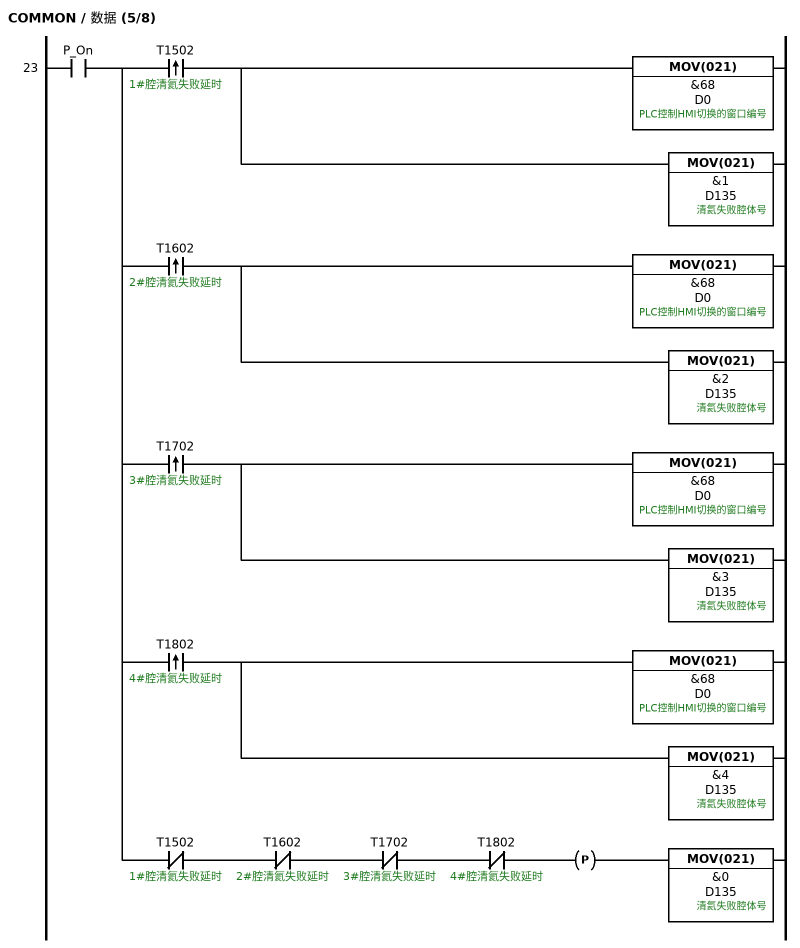
; [picture p432: COMMON / 数据, rungs 23-23]
; rung 23
LD P_On
OUT TR0
@AND T1502  ; 1#腔清氦失败延时
MOV(021) &68 D0  ; PLC控制HMI切换的窗口编号
MOV(021) &1 D135  ; 清氦失败腔体号
LD TR0
@AND T1602  ; 2#腔清氦失败延时
MOV(021) &68 D0  ; PLC控制HMI切换的窗口编号
MOV(021) &2 D135  ; 清氦失败腔体号
LD TR0
@AND T1702  ; 3#腔清氦失败延时
MOV(021) &68 D0  ; PLC控制HMI切换的窗口编号
MOV(021) &3 D135  ; 清氦失败腔体号
LD TR0
@AND T1802  ; 4#腔清氦失败延时
MOV(021) &68 D0  ; PLC控制HMI切换的窗口编号
MOV(021) &4 D135  ; 清氦失败腔体号
LD TR0
ANDNOT T1502  ; 1#腔清氦失败延时
ANDNOT T1602  ; 2#腔清氦失败延时
ANDNOT T1702  ; 3#腔清氦失败延时
ANDNOT T1802  ; 4#腔清氦失败延时
UP(521)
MOV(021) &0 D135  ; 清氦失败腔体号

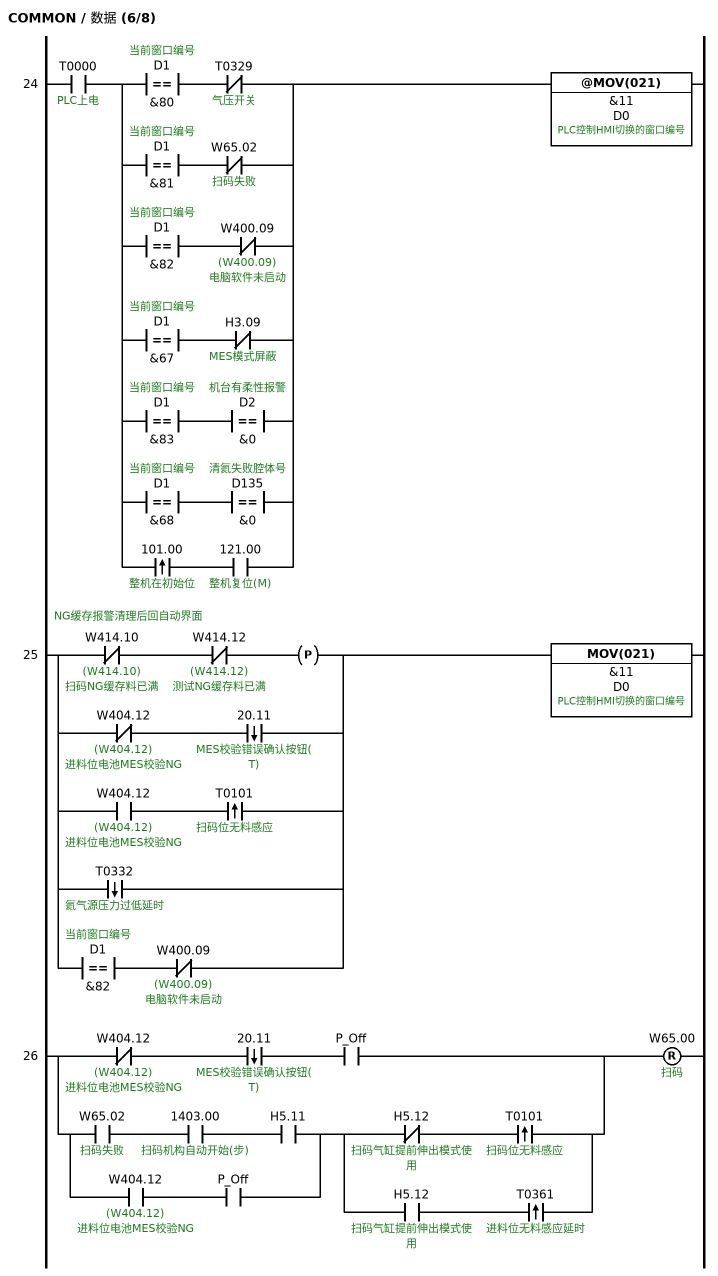
; rung 24
LD T0000  ; PLC上电
LD=(300) D1 &80  ; 当前窗口编号
ANDNOT T0329  ; 气压开关
LD=(300) D1 &81  ; 当前窗口编号
ANDNOT W65.02  ; 扫码失败
ORLD
LD=(300) D1 &82  ; 当前窗口编号
ANDNOT W400.09  ; (W400.09) 电脑软件未启动
ORLD
LD=(300) D1 &67  ; 当前窗口编号
ANDNOT H3.09  ; MES模式屏蔽
ORLD
LD=(300) D1 &83  ; 当前窗口编号
AND=(300) D2 &0  ; 机台有柔性报警
ORLD
LD=(300) D1 &68  ; 当前窗口编号
AND=(300) D135 &0  ; 清氦失败腔体号
ORLD
@LD 101.00  ; 整机在初始位
AND 121.00  ; 整机复位(M)
ORLD
ANDLD
@MOV(021) &11 D0  ; PLC控制HMI切换的窗口编号
; rung 25: NG缓存报警清理后回自动界面
LDNOT W414.10  ; (W414.10) 扫码NG缓存料已满
ANDNOT W414.12  ; (W414.12) 测试NG缓存料已满
UP(521)
LDNOT W404.12  ; (W404.12) 进料位电池MES校验NG
%AND 20.11  ; MES校验错误确认按钮(T)
ORLD
LD W404.12  ; (W404.12) 进料位电池MES校验NG
@AND T0101  ; 扫码位无料感应
ORLD
%OR T0332  ; 氦气源压力过低延时
LD=(300) D1 &82  ; 当前窗口编号
ANDNOT W400.09  ; (W400.09) 电脑软件未启动
ORLD
MOV(021) &11 D0  ; PLC控制HMI切换的窗口编号
; rung 26
LDNOT W404.12  ; (W404.12) 进料位电池MES校验NG
%AND 20.11  ; MES校验错误确认按钮(T)
AND P_Off
LD W65.02  ; 扫码失败
AND 1403.00  ; 扫码机构自动开始(步)
AND H5.11
LD W404.12  ; (W404.12) 进料位电池MES校验NG
AND P_Off
ORLD
LDNOT H5.12  ; 扫码气缸提前伸出模式使用
@AND T0101  ; 扫码位无料感应
LD H5.12  ; 扫码气缸提前伸出模式使用
@AND T0361  ; 进料位无料感应延时
ORLD
ANDLD
ORLD
RSET W65.00  ; 扫码

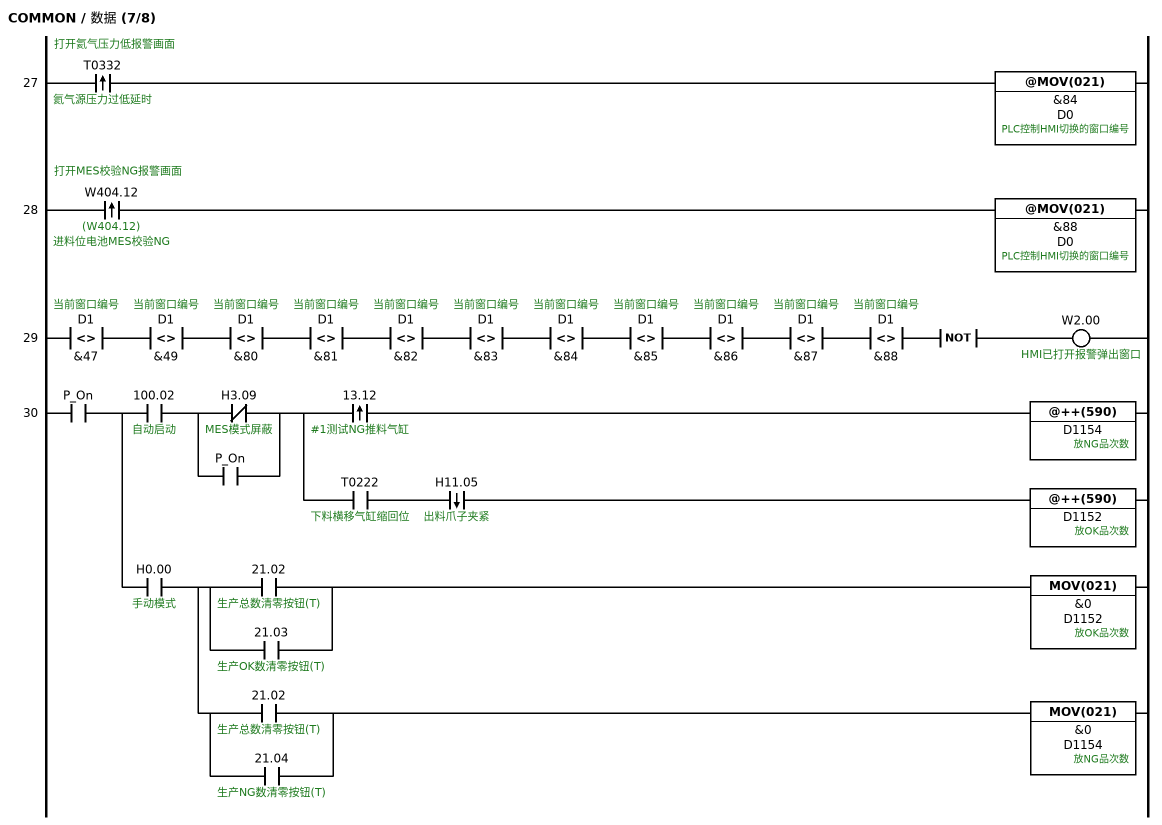
; rung 27: 打开氦气压力低报警画面
@LD T0332  ; 氦气源压力过低延时
@MOV(021) &84 D0  ; PLC控制HMI切换的窗口编号
; rung 28: 打开MES校验NG报警画面
@LD W404.12  ; (W404.12) 进料位电池MES校验NG
@MOV(021) &88 D0  ; PLC控制HMI切换的窗口编号
; rung 29
LD<>(305) D1 &47  ; 当前窗口编号
AND<>(305) D1 &49  ; 当前窗口编号
AND<>(305) D1 &80  ; 当前窗口编号
AND<>(305) D1 &81  ; 当前窗口编号
AND<>(305) D1 &82  ; 当前窗口编号
AND<>(305) D1 &83  ; 当前窗口编号
AND<>(305) D1 &84  ; 当前窗口编号
AND<>(305) D1 &85  ; 当前窗口编号
AND<>(305) D1 &86  ; 当前窗口编号
AND<>(305) D1 &87  ; 当前窗口编号
AND<>(305) D1 &88  ; 当前窗口编号
NOT(520)
OUT W2.00  ; HMI已打开报警弹出窗口
; rung 30
LD P_On
OUT TR0
AND 100.02  ; 自动启动
LDNOT H3.09  ; MES模式屏蔽
OR P_On
ANDLD
OUT TR1
@AND 13.12  ; #1测试NG推料气缸
@++(590) D1154  ; 放NG品次数
LD TR1
AND T0222  ; 下料横移气缸缩回位
%AND H11.05  ; 出料爪子夹紧
@++(590) D1152  ; 放OK品次数
LD TR0
AND H0.00  ; 手动模式
OUT TR0
LD 21.02  ; 生产总数清零按钮(T)
OR 21.03  ; 生产OK数清零按钮(T)
ANDLD
MOV(021) &0 D1152  ; 放OK品次数
LD TR0
LD 21.02  ; 生产总数清零按钮(T)
OR 21.04  ; 生产NG数清零按钮(T)
ANDLD
MOV(021) &0 D1154  ; 放NG品次数

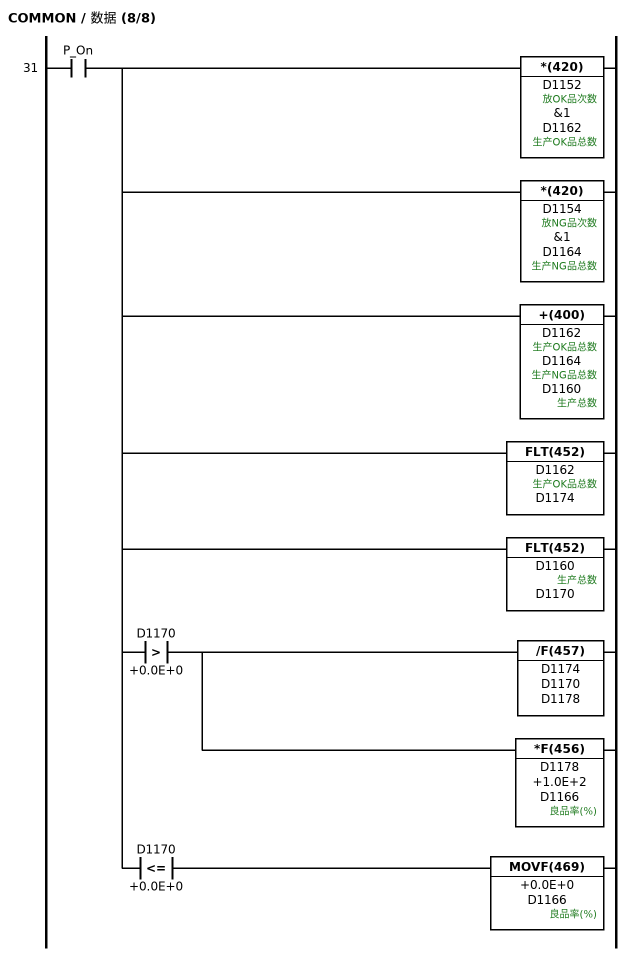
; rung 31
LD P_On
OUT TR0
*(420) D1152 &1 D1162  ; 放OK品次数, 生产OK品总数
*(420) D1154 &1 D1164  ; 放NG品次数, 生产NG品总数
+(400) D1162 D1164 D1160  ; 生产OK品总数, 生产NG品总数, 生产总数
FLT(452) D1162 D1174  ; 生产OK品总数
FLT(452) D1160 D1170  ; 生产总数
AND>F(333) D1170 +0.0E+0
/F(457) D1174 D1170 D1178
*F(456) D1178 +1.0E+2 D1166  ; 良品率(%)
LD TR0
AND<=F(332) D1170 +0.0E+0
MOVF(469) +0.0E+0 D1166  ; 良品率(%)

### Section 报警

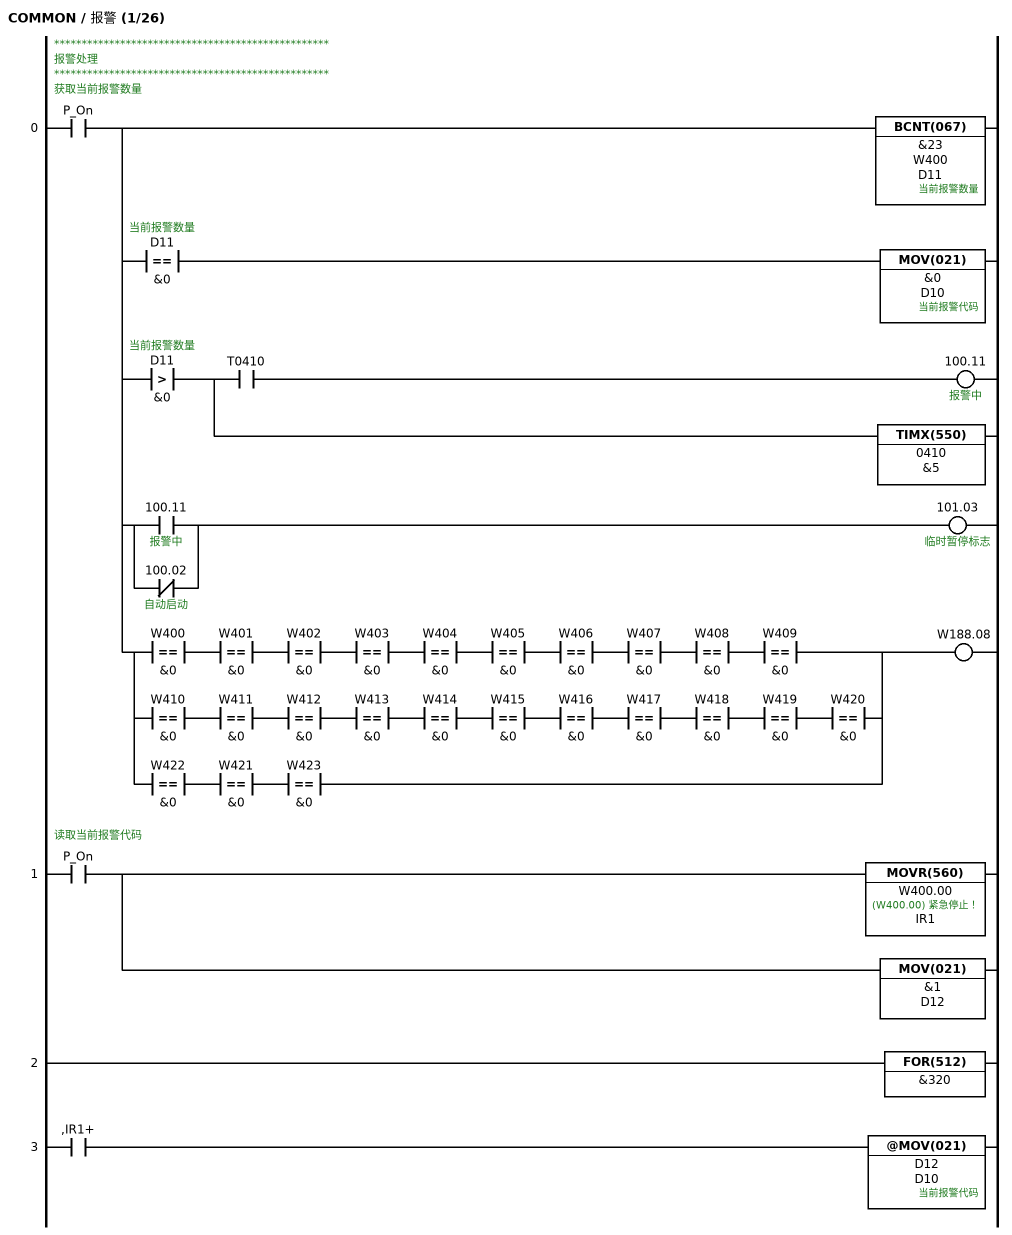
; rung 0: ************************************************** / 报警处理 / ************************************************** / 获取当前报警数量
LD P_On
OUT TR0
BCNT(067) &23 W400 D11  ; 当前报警数量
AND=(300) D11 &0  ; 当前报警数量
MOV(021) &0 D10  ; 当前报警代码
LD TR0
AND>(320) D11 &0  ; 当前报警数量
OUT TR1
AND T0410
OUT 100.11  ; 报警中
LD TR1
TIMX(550) 0410 &5
LD TR0
LD 100.11  ; 报警中
ORNOT 100.02  ; 自动启动
ANDLD
OUT 101.03  ; 临时暂停标志
LD TR0
LD=(300) W400 &0
AND=(300) W401 &0
AND=(300) W402 &0
AND=(300) W403 &0
AND=(300) W404 &0
AND=(300) W405 &0
AND=(300) W406 &0
AND=(300) W407 &0
AND=(300) W408 &0
AND=(300) W409 &0
LD=(300) W410 &0
AND=(300) W411 &0
AND=(300) W412 &0
AND=(300) W413 &0
AND=(300) W414 &0
AND=(300) W415 &0
AND=(300) W416 &0
AND=(300) W417 &0
AND=(300) W418 &0
AND=(300) W419 &0
AND=(300) W420 &0
ORLD
LD=(300) W422 &0
AND=(300) W421 &0
AND=(300) W423 &0
ORLD
ANDLD
OUT W188.08
; rung 1: 读取当前报警代码
LD P_On
MOVR(560) W400.00 IR1  ; (W400.00) 紧急停止！
MOV(021) &1 D12
; rung 2
FOR(512) &320
; rung 3
LD ,IR1+
@MOV(021) D12 D10  ; 当前报警代码

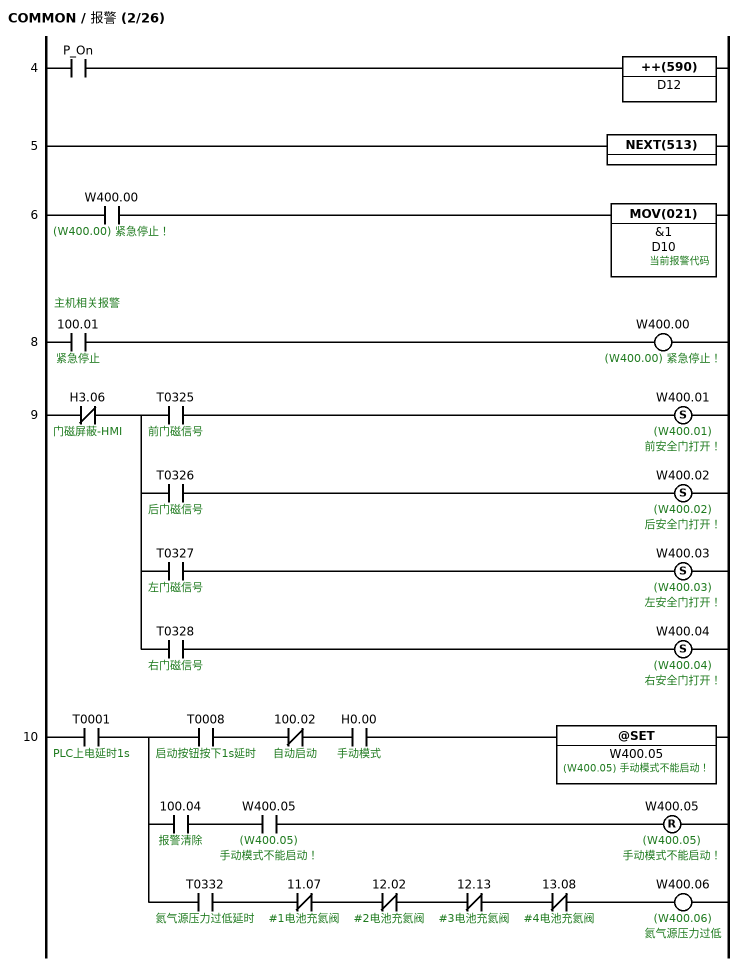
; rung 4
LD P_On
++(590) D12
; rung 5
NEXT(513)
; rung 6
LD W400.00  ; (W400.00) 紧急停止！
MOV(021) &1 D10  ; 当前报警代码
; rung 7: ************************************************************************** / 报警处理 / **************************************************************************
; rung 8: 主机相关报警
LD 100.01  ; 紧急停止
OUT W400.00  ; (W400.00) 紧急停止！
; rung 9
LDNOT H3.06  ; 门磁屏蔽-HMI
OUT TR0
AND T0325  ; 前门磁信号
SET W400.01  ; (W400.01) 前安全门打开！
LD TR0
AND T0326  ; 后门磁信号
SET W400.02  ; (W400.02) 后安全门打开！
LD TR0
AND T0327  ; 左门磁信号
SET W400.03  ; (W400.03) 左安全门打开！
LD TR0
AND T0328  ; 右门磁信号
SET W400.04  ; (W400.04) 右安全门打开！
; rung 10
LD T0001  ; PLC上电延时1s
OUT TR0
AND T0008  ; 启动按钮按下1s延时
ANDNOT 100.02  ; 自动启动
AND H0.00  ; 手动模式
@SET W400.05  ; (W400.05) 手动模式不能启动！
LD TR0
AND 100.04  ; 报警清除
AND W400.05  ; (W400.05) 手动模式不能启动！
RSET W400.05  ; (W400.05) 手动模式不能启动！
LD TR0
AND T0332  ; 氦气源压力过低延时
ANDNOT 11.07  ; #1电池充氦阀
ANDNOT 12.02  ; #2电池充氦阀
ANDNOT 12.13  ; #3电池充氦阀
ANDNOT 13.08  ; #4电池充氦阀
OUT W400.06  ; (W400.06) 氦气源压力过低

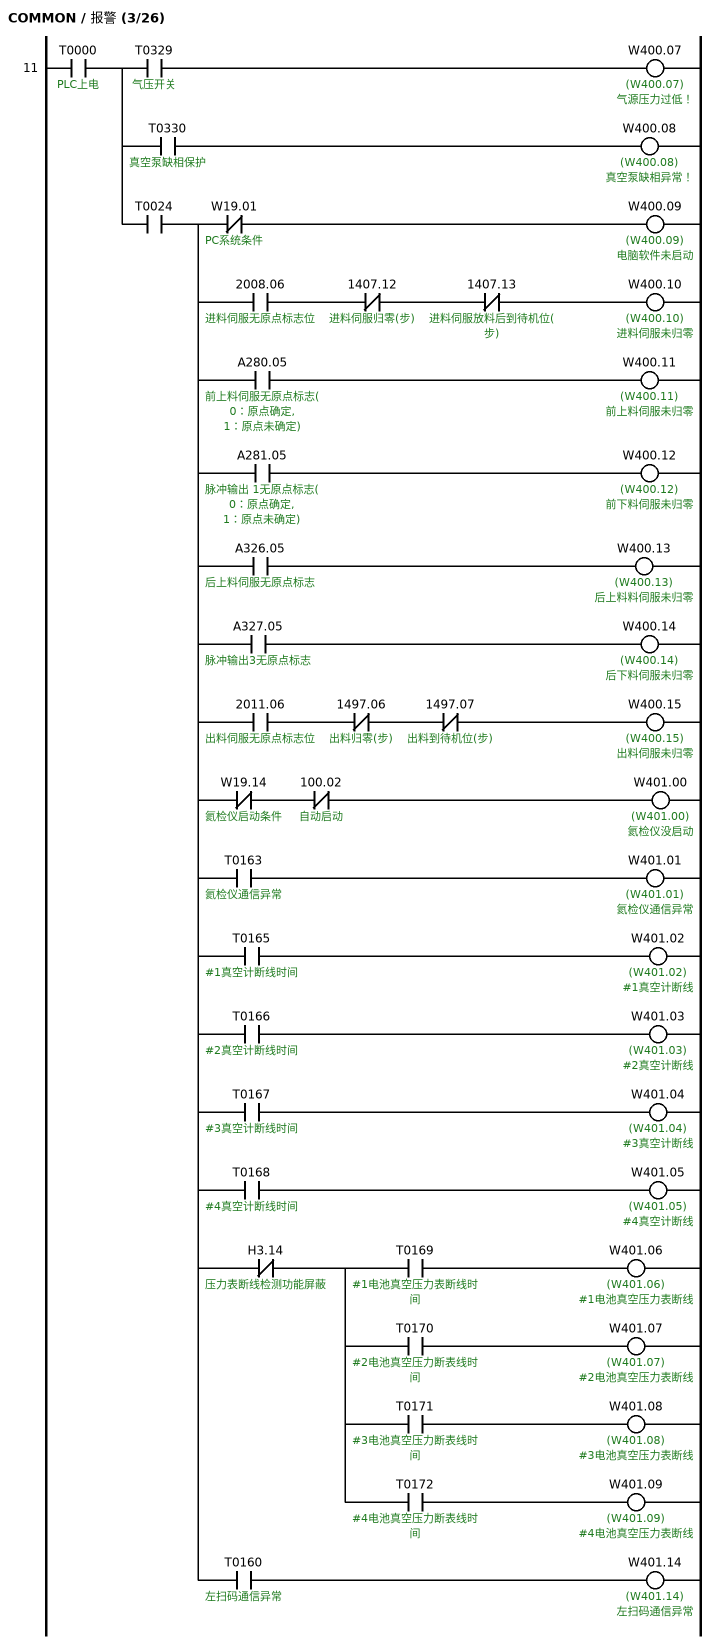
; rung 11
LD T0000  ; PLC上电
OUT TR0
AND T0329  ; 气压开关
OUT W400.07  ; (W400.07) 气源压力过低！
LD TR0
AND T0330  ; 真空泵缺相保护
OUT W400.08  ; (W400.08) 真空泵缺相异常！
LD TR0
AND T0024
OUT TR0
ANDNOT W19.01  ; PC系统条件
OUT W400.09  ; (W400.09) 电脑软件未启动
LD TR0
AND 2008.06  ; 进料伺服无原点标志位
ANDNOT 1407.12  ; 进料伺服归零(步)
ANDNOT 1407.13  ; 进料伺服放料后到待机位(步)
OUT W400.10  ; (W400.10) 进料伺服未归零
LD TR0
AND A280.05  ; 前上料伺服无原点标志(0：原点确定,1：原点未确定)
OUT W400.11  ; (W400.11) 前上料伺服未归零
LD TR0
AND A281.05  ; 脉冲输出 1无原点标志(0：原点确定,1：原点未确定)
OUT W400.12  ; (W400.12) 前下料伺服未归零
LD TR0
AND A326.05  ; 后上料伺服无原点标志
OUT W400.13  ; (W400.13) 后上料料伺服未归零
LD TR0
AND A327.05  ; 脉冲输出3无原点标志
OUT W400.14  ; (W400.14) 后下料伺服未归零
LD TR0
AND 2011.06  ; 出料伺服无原点标志位
ANDNOT 1497.06  ; 出料归零(步)
ANDNOT 1497.07  ; 出料到待机位(步)
OUT W400.15  ; (W400.15) 出料伺服未归零
LD TR0
ANDNOT W19.14  ; 氦检仪启动条件
ANDNOT 100.02  ; 自动启动
OUT W401.00  ; (W401.00) 氦检仪没启动
LD TR0
AND T0163  ; 氦检仪通信异常
OUT W401.01  ; (W401.01) 氦检仪通信异常
LD TR0
AND T0165  ; #1真空计断线时间
OUT W401.02  ; (W401.02) #1真空计断线
LD TR0
AND T0166  ; #2真空计断线时间
OUT W401.03  ; (W401.03) #2真空计断线
LD TR0
AND T0167  ; #3真空计断线时间
OUT W401.04  ; (W401.04) #3真空计断线
LD TR0
AND T0168  ; #4真空计断线时间
OUT W401.05  ; (W401.05) #4真空计断线
LD TR0
ANDNOT H3.14  ; 压力表断线检测功能屏蔽
OUT TR1
AND T0169  ; #1电池真空压力表断线时间
OUT W401.06  ; (W401.06) #1电池真空压力表断线
LD TR1
AND T0170  ; #2电池真空压力断表线时间
OUT W401.07  ; (W401.07) #2电池真空压力表断线
LD TR1
AND T0171  ; #3电池真空压力断表线时间
OUT W401.08  ; (W401.08) #3电池真空压力表断线
LD TR1
AND T0172  ; #4电池真空压力断表线时间
OUT W401.09  ; (W401.09) #4电池真空压力表断线
LD TR0
AND T0160  ; 左扫码通信异常
OUT W401.14  ; (W401.14) 左扫码通信异常

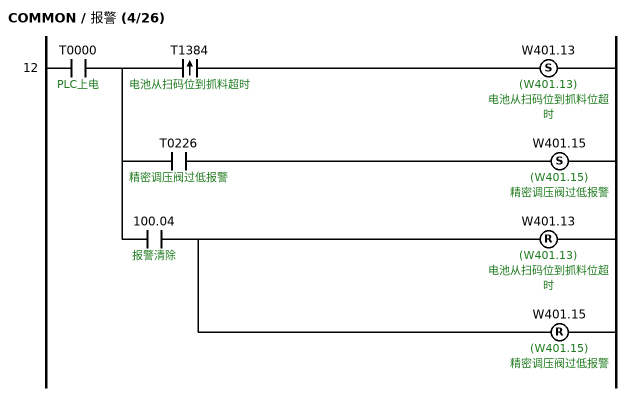
; rung 12
LD T0000  ; PLC上电
OUT TR0
@AND T1384  ; 电池从扫码位到抓料超时
SET W401.13  ; (W401.13) 电池从扫码位到抓料位超时
LD TR0
AND T0226  ; 精密调压阀过低报警
SET W401.15  ; (W401.15) 精密调压阀过低报警
LD TR0
AND 100.04  ; 报警清除
RSET W401.13  ; (W401.13) 电池从扫码位到抓料位超时
RSET W401.15  ; (W401.15) 精密调压阀过低报警

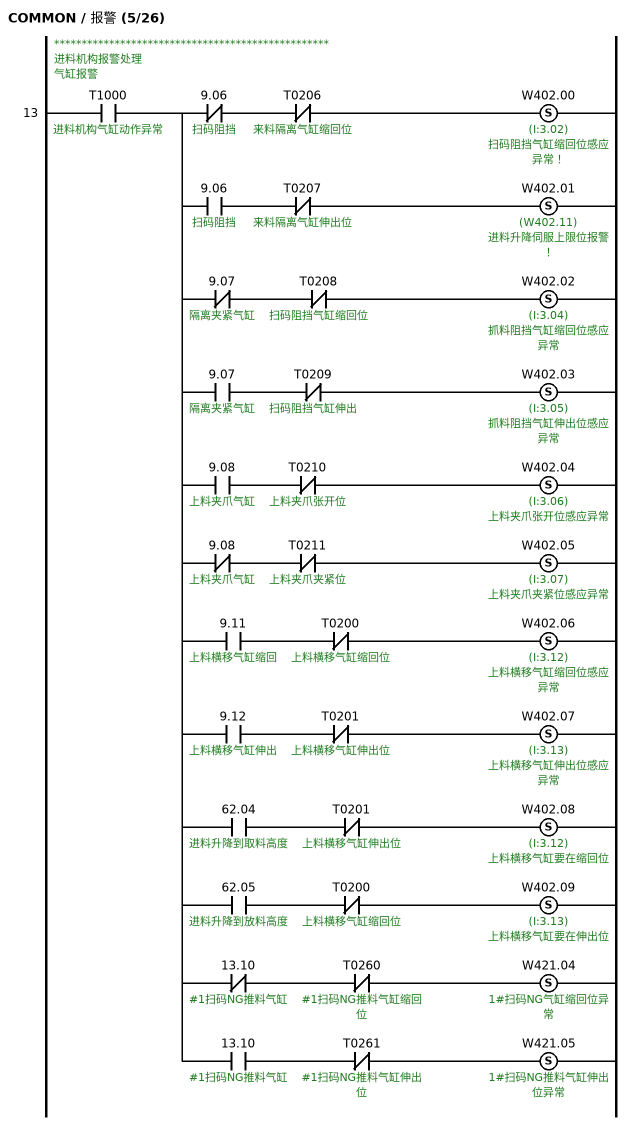
; rung 13: ************************************************** / 进料机构报警处理 / 气缸报警
LD T1000  ; 进料机构气缸动作异常
OUT TR0
ANDNOT 9.06  ; 扫码阻挡
ANDNOT T0206  ; 来料隔离气缸缩回位
SET W402.00  ; (I:3.02) 扫码阻挡气缸缩回位感应异常！
LD TR0
AND 9.06  ; 扫码阻挡
ANDNOT T0207  ; 来料隔离气缸伸出位
SET W402.01  ; (W402.11) 进料升降伺服上限位报警！
LD TR0
ANDNOT 9.07  ; 隔离夹紧气缸
ANDNOT T0208  ; 扫码阻挡气缸缩回位
SET W402.02  ; (I:3.04) 抓料阻挡气缸缩回位感应异常
LD TR0
AND 9.07  ; 隔离夹紧气缸
ANDNOT T0209  ; 扫码阻挡气缸伸出
SET W402.03  ; (I:3.05) 抓料阻挡气缸伸出位感应异常
LD TR0
AND 9.08  ; 上料夹爪气缸
ANDNOT T0210  ; 上料夹爪张开位
SET W402.04  ; (I:3.06) 上料夹爪张开位感应异常
LD TR0
ANDNOT 9.08  ; 上料夹爪气缸
ANDNOT T0211  ; 上料夹爪夹紧位
SET W402.05  ; (I:3.07) 上料夹爪夹紧位感应异常
LD TR0
AND 9.11  ; 上料横移气缸缩回
ANDNOT T0200  ; 上料横移气缸缩回位
SET W402.06  ; (I:3.12) 上料横移气缸缩回位感应异常
LD TR0
AND 9.12  ; 上料横移气缸伸出
ANDNOT T0201  ; 上料横移气缸伸出位
SET W402.07  ; (I:3.13) 上料横移气缸伸出位感应异常
LD TR0
AND 62.04  ; 进料升降到取料高度
ANDNOT T0201  ; 上料横移气缸伸出位
SET W402.08  ; (I:3.12) 上料横移气缸要在缩回位
LD TR0
AND 62.05  ; 进料升降到放料高度
ANDNOT T0200  ; 上料横移气缸缩回位
SET W402.09  ; (I:3.13) 上料横移气缸要在伸出位
LD TR0
ANDNOT 13.10  ; #1扫码NG推料气缸
ANDNOT T0260  ; #1扫码NG推料气缸缩回位
SET W421.04  ; 1#扫码NG气缸缩回位异常
LD TR0
AND 13.10  ; #1扫码NG推料气缸
ANDNOT T0261  ; #1扫码NG推料气缸伸出位
SET W421.05  ; 1#扫码NG推料气缸伸出位异常

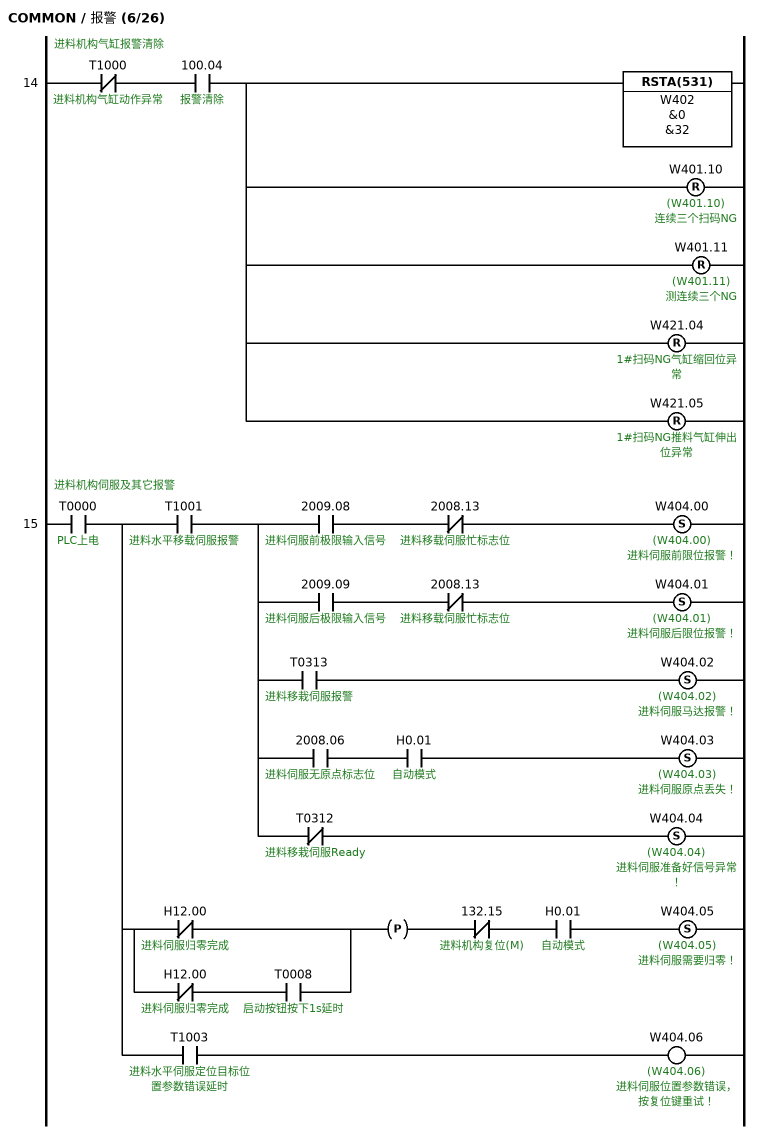
; rung 14: 进料机构气缸报警清除
LDNOT T1000  ; 进料机构气缸动作异常
AND 100.04  ; 报警清除
RSTA(531) W402 &0 &32
RSET W401.10  ; (W401.10) 连续三个扫码NG
RSET W401.11  ; (W401.11) 测连续三个NG
RSET W421.04  ; 1#扫码NG气缸缩回位异常
RSET W421.05  ; 1#扫码NG推料气缸伸出位异常
; rung 15: 进料机构伺服及其它报警
LD T0000  ; PLC上电
OUT TR0
AND T1001  ; 进料水平移载伺服报警
OUT TR1
AND 2009.08  ; 进料伺服前极限输入信号
ANDNOT 2008.13  ; 进料移载伺服忙标志位
SET W404.00  ; (W404.00) 进料伺服前限位报警！
LD TR1
AND 2009.09  ; 进料伺服后极限输入信号
ANDNOT 2008.13  ; 进料移载伺服忙标志位
SET W404.01  ; (W404.01) 进料伺服后限位报警！
LD TR1
AND T0313  ; 进料移栽伺服报警
SET W404.02  ; (W404.02) 进料伺服马达报警！
LD TR1
AND 2008.06  ; 进料伺服无原点标志位
AND H0.01  ; 自动模式
SET W404.03  ; (W404.03) 进料伺服原点丢失！
LD TR1
ANDNOT T0312  ; 进料移栽伺服Ready
SET W404.04  ; (W404.04) 进料伺服准备好信号异常！
LD TR0
LDNOT H12.00  ; 进料伺服归零完成
LDNOT H12.00  ; 进料伺服归零完成
AND T0008  ; 启动按钮按下1s延时
ORLD
ANDLD
UP(521)
ANDNOT 132.15  ; 进料机构复位(M)
AND H0.01  ; 自动模式
SET W404.05  ; (W404.05) 进料伺服需要归零！
LD TR0
AND T1003  ; 进料水平伺服定位目标位置参数错误延时
OUT W404.06  ; (W404.06) 进料伺服位置参数错误，按复位键重试！

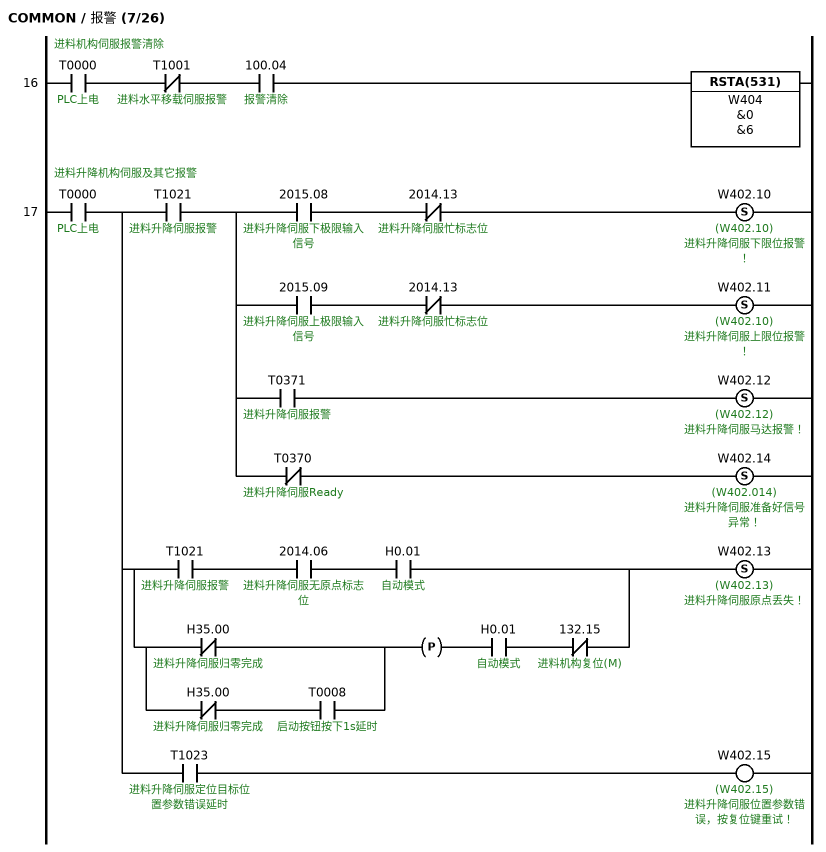
; rung 16: 进料机构伺服报警清除
LD T0000  ; PLC上电
ANDNOT T1001  ; 进料水平移载伺服报警
AND 100.04  ; 报警清除
RSTA(531) W404 &0 &6
; rung 17: 进料升降机构伺服及其它报警
LD T0000  ; PLC上电
OUT TR0
AND T1021  ; 进料升降伺服报警
OUT TR1
AND 2015.08  ; 进料升降伺服下极限输入信号
ANDNOT 2014.13  ; 进料升降伺服忙标志位
SET W402.10  ; (W402.10) 进料升降伺服下限位报警！
LD TR1
AND 2015.09  ; 进料升降伺服上极限输入信号
ANDNOT 2014.13  ; 进料升降伺服忙标志位
SET W402.11  ; (W402.10) 进料升降伺服上限位报警！
LD TR1
AND T0371  ; 进料升降伺服报警
SET W402.12  ; (W402.12) 进料升降伺服马达报警！
LD TR1
ANDNOT T0370  ; 进料升降伺服Ready
SET W402.14  ; (W402.014) 进料升降伺服准备好信号异常！
LD TR0
LD T1021  ; 进料升降伺服报警
AND 2014.06  ; 进料升降伺服无原点标志位
AND H0.01  ; 自动模式
LDNOT H35.00  ; 进料升降伺服归零完成
LDNOT H35.00  ; 进料升降伺服归零完成
AND T0008  ; 启动按钮按下1s延时
ORLD
UP(521)
AND H0.01  ; 自动模式
ANDNOT 132.15  ; 进料机构复位(M)
ORLD
ANDLD
SET W402.13  ; (W402.13) 进料升降伺服原点丢失！
LD TR0
AND T1023  ; 进料升降伺服定位目标位置参数错误延时
OUT W402.15  ; (W402.15) 进料升降伺服位置参数错误，按复位键重试！

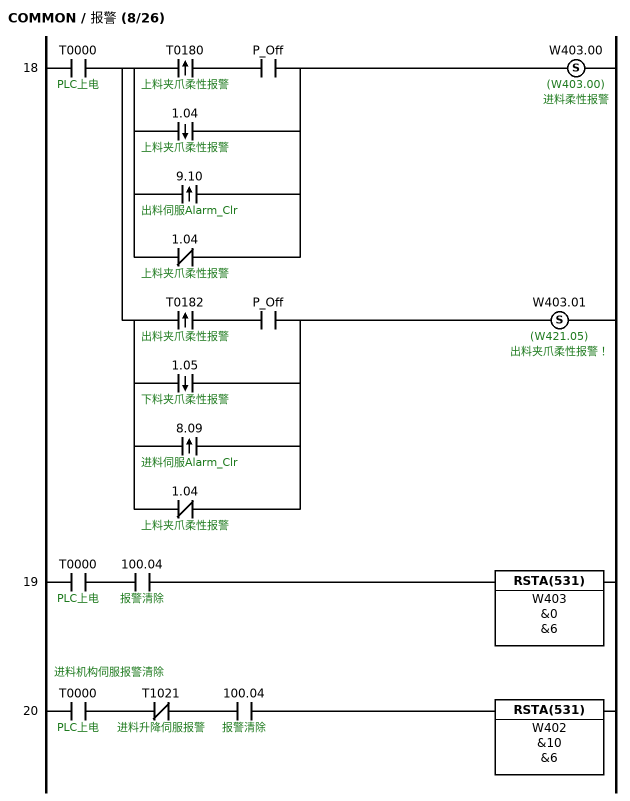
; rung 18
LD T0000  ; PLC上电
OUT TR0
@LD T0180  ; 上料夹爪柔性报警
AND P_Off
%OR 1.04  ; 上料夹爪柔性报警
@OR 9.10  ; 出料伺服Alarm_Clr
ORNOT 1.04  ; 上料夹爪柔性报警
ANDLD
SET W403.00  ; (W403.00) 进料柔性报警
LD TR0
@LD T0182  ; 出料夹爪柔性报警
AND P_Off
%OR 1.05  ; 下料夹爪柔性报警
@OR 8.09  ; 进料伺服Alarm_Clr
ORNOT 1.04  ; 上料夹爪柔性报警
ANDLD
SET W403.01  ; (W421.05) 出料夹爪柔性报警！
; rung 19
LD T0000  ; PLC上电
AND 100.04  ; 报警清除
RSTA(531) W403 &0 &6
; rung 20: 进料机构伺服报警清除
LD T0000  ; PLC上电
ANDNOT T1021  ; 进料升降伺服报警
AND 100.04  ; 报警清除
RSTA(531) W402 &10 &6

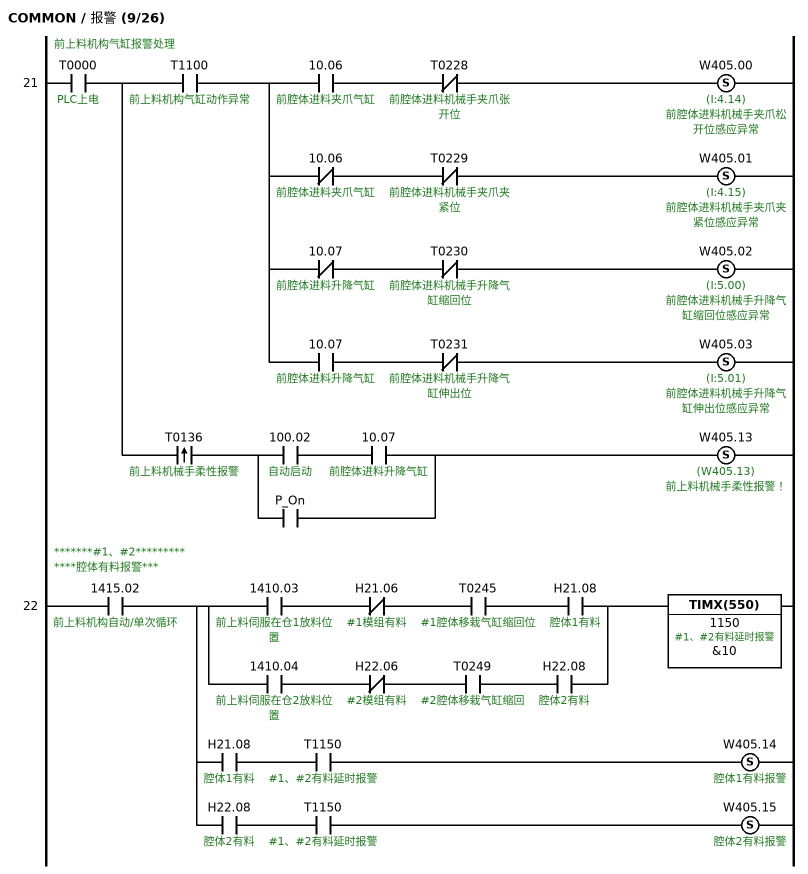
; rung 21: 前上料机构气缸报警处理
LD T0000  ; PLC上电
OUT TR0
AND T1100  ; 前上料机构气缸动作异常
OUT TR1
AND 10.06  ; 前腔体进料夹爪气缸
ANDNOT T0228  ; 前腔体进料机械手夹爪张开位
SET W405.00  ; (I:4.14) 前腔体进料机械手夹爪松开位感应异常
LD TR1
ANDNOT 10.06  ; 前腔体进料夹爪气缸
ANDNOT T0229  ; 前腔体进料机械手夹爪夹紧位
SET W405.01  ; (I:4.15) 前腔体进料机械手夹爪夹紧位感应异常
LD TR1
ANDNOT 10.07  ; 前腔体进料升降气缸
ANDNOT T0230  ; 前腔体进料机械手升降气缸缩回位
SET W405.02  ; (I:5.00) 前腔体进料机械手升降气缸缩回位感应异常
LD TR1
AND 10.07  ; 前腔体进料升降气缸
ANDNOT T0231  ; 前腔体进料机械手升降气缸伸出位
SET W405.03  ; (I:5.01) 前腔体进料机械手升降气缸伸出位感应异常
LD TR0
!@AND T0136  ; 前上料机械手柔性报警
LD 100.02  ; 自动启动
AND 10.07  ; 前腔体进料升降气缸
OR P_On
ANDLD
SET W405.13  ; (W405.13) 前上料机械手柔性报警！
; rung 22: *******#1、#2********* / ****腔体有料报警***
LD 1415.02  ; 前上料机构自动/单次循环
OUT TR0
LD 1410.03  ; 前上料伺服在仓1放料位置
ANDNOT H21.06  ; #1模组有料
AND T0245  ; #1腔体移栽气缸缩回位
AND H21.08  ; 腔体1有料
LD 1410.04  ; 前上料伺服在仓2放料位置
ANDNOT H22.06  ; #2模组有料
AND T0249  ; #2腔体移栽气缸缩回
AND H22.08  ; 腔体2有料
ORLD
ANDLD
TIMX(550) 1150 &10  ; #1、#2有料延时报警
LD TR0
AND H21.08  ; 腔体1有料
AND T1150  ; #1、#2有料延时报警
SET W405.14  ; 腔体1有料报警
LD TR0
AND H22.08  ; 腔体2有料
AND T1150  ; #1、#2有料延时报警
SET W405.15  ; 腔体2有料报警

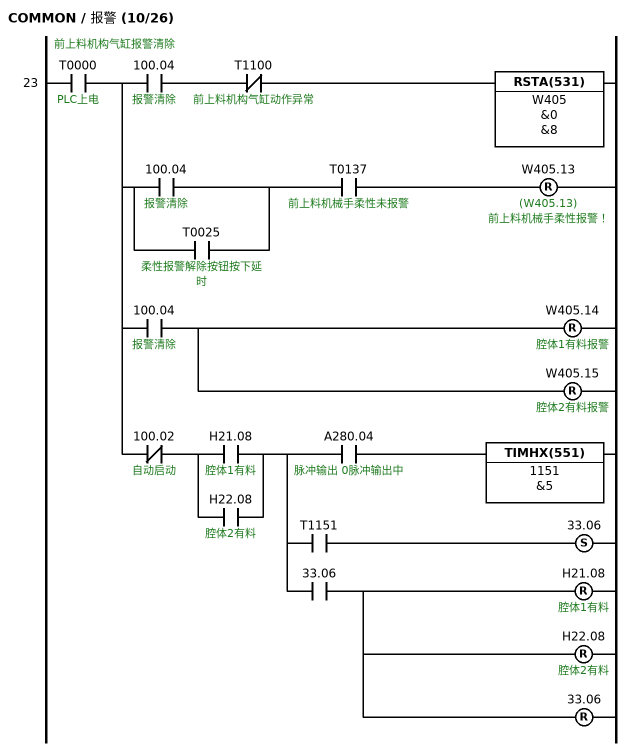
; rung 23: 前上料机构气缸报警清除
LD T0000  ; PLC上电
OUT TR0
AND 100.04  ; 报警清除
ANDNOT T1100  ; 前上料机构气缸动作异常
RSTA(531) W405 &0 &8
LD TR0
LD 100.04  ; 报警清除
OR T0025  ; 柔性报警解除按钮按下延时
ANDLD
AND T0137  ; 前上料机械手柔性未报警
RSET W405.13  ; (W405.13) 前上料机械手柔性报警！
LD TR0
AND 100.04  ; 报警清除
RSET W405.14  ; 腔体1有料报警
RSET W405.15  ; 腔体2有料报警
LD TR0
ANDNOT 100.02  ; 自动启动
LD H21.08  ; 腔体1有料
OR H22.08  ; 腔体2有料
ANDLD
OUT TR0
AND A280.04  ; 脉冲输出 0脉冲输出中
TIMHX(551) 1151 &5
LD TR0
AND T1151
SET 33.06
LD TR0
AND 33.06
RSET H21.08  ; 腔体1有料
RSET H22.08  ; 腔体2有料
RSET 33.06

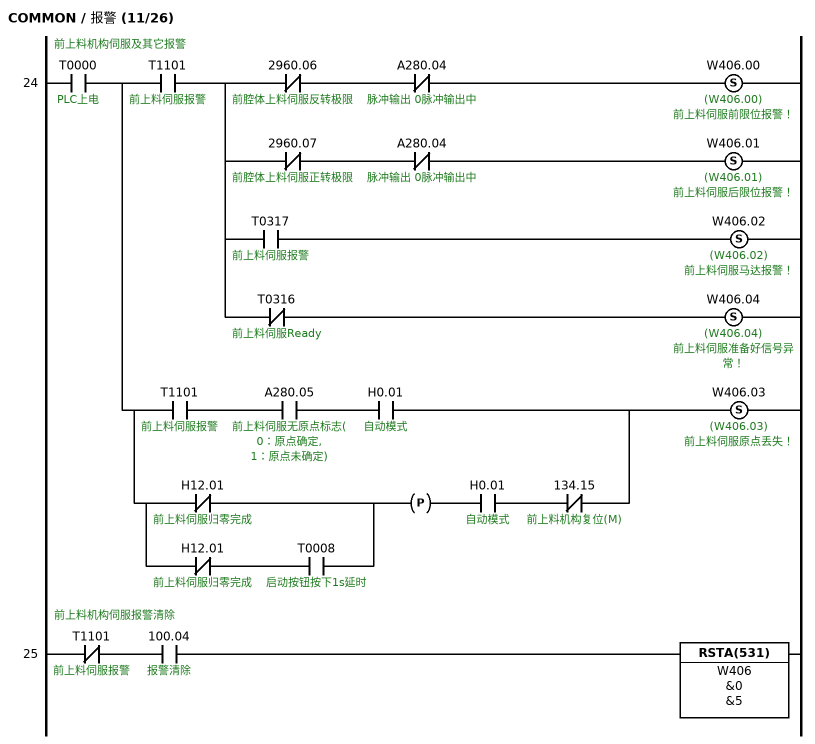
; rung 24: 前上料机构伺服及其它报警
LD T0000  ; PLC上电
OUT TR0
AND T1101  ; 前上料伺服报警
OUT TR1
ANDNOT 2960.06  ; 前腔体上料伺服反转极限
ANDNOT A280.04  ; 脉冲输出 0脉冲输出中
SET W406.00  ; (W406.00) 前上料伺服前限位报警！
LD TR1
ANDNOT 2960.07  ; 前腔体上料伺服正转极限
ANDNOT A280.04  ; 脉冲输出 0脉冲输出中
SET W406.01  ; (W406.01) 前上料伺服后限位报警！
LD TR1
AND T0317  ; 前上料伺服报警
SET W406.02  ; (W406.02) 前上料伺服马达报警！
LD TR1
ANDNOT T0316  ; 前上料伺服Ready
SET W406.04  ; (W406.04) 前上料伺服准备好信号异常！
LD TR0
LD T1101  ; 前上料伺服报警
AND A280.05  ; 前上料伺服无原点标志(0：原点确定,1：原点未确定)
AND H0.01  ; 自动模式
LDNOT H12.01  ; 前上料伺服归零完成
LDNOT H12.01  ; 前上料伺服归零完成
AND T0008  ; 启动按钮按下1s延时
ORLD
UP(521)
AND H0.01  ; 自动模式
ANDNOT 134.15  ; 前上料机构复位(M)
ORLD
ANDLD
SET W406.03  ; (W406.03) 前上料伺服原点丢失！
; rung 25: 前上料机构伺服报警清除
LDNOT T1101  ; 前上料伺服报警
AND 100.04  ; 报警清除
RSTA(531) W406 &0 &5

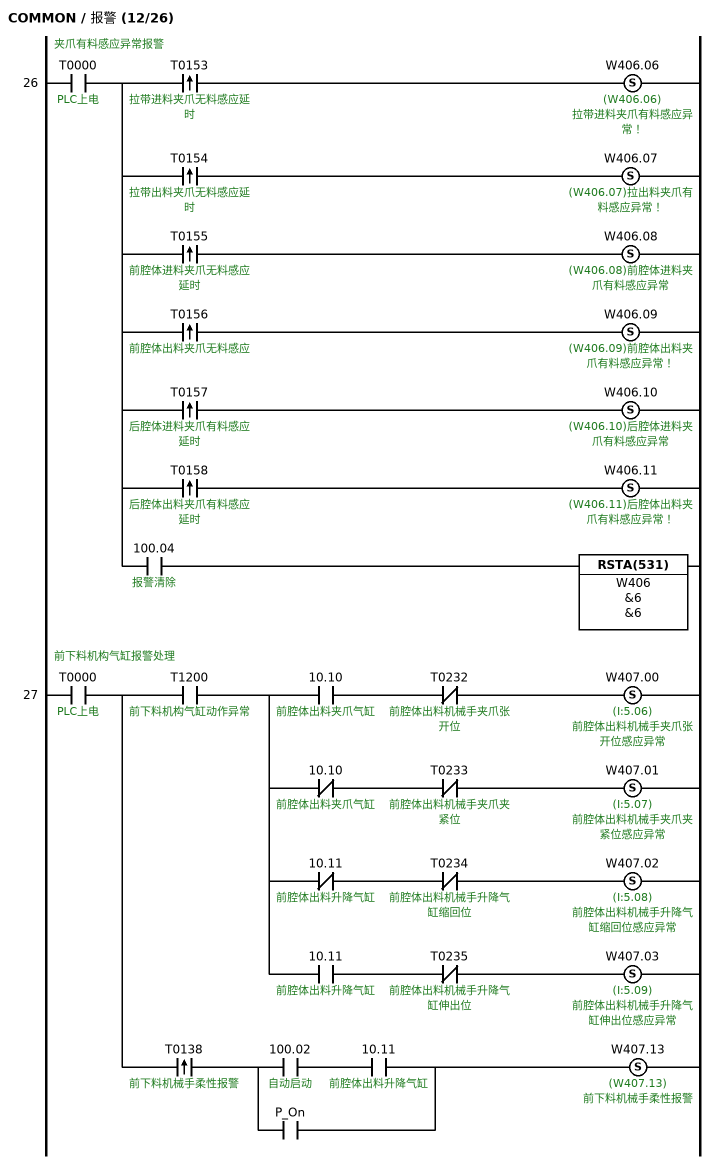
; rung 26: 夹爪有料感应异常报警
LD T0000  ; PLC上电
OUT TR0
@AND T0153  ; 拉带进料夹爪无料感应延时
SET W406.06  ; (W406.06) 拉带进料夹爪有料感应异常！
LD TR0
@AND T0154  ; 拉带出料夹爪无料感应延时
SET W406.07  ; (W406.07)拉出料夹爪有料感应异常！
LD TR0
@AND T0155  ; 前腔体进料夹爪无料感应延时
SET W406.08  ; (W406.08)前腔体进料夹爪有料感应异常
LD TR0
@AND T0156  ; 前腔体出料夹爪无料感应
SET W406.09  ; (W406.09)前腔体出料夹爪有料感应异常！
LD TR0
@AND T0157  ; 后腔体进料夹爪有料感应延时
SET W406.10  ; (W406.10)后腔体进料夹爪有料感应异常
LD TR0
@AND T0158  ; 后腔体出料夹爪有料感应延时
SET W406.11  ; (W406.11)后腔体出料夹爪有料感应异常！
LD TR0
AND 100.04  ; 报警清除
RSTA(531) W406 &6 &6
; rung 27: 前下料机构气缸报警处理
LD T0000  ; PLC上电
OUT TR0
AND T1200  ; 前下料机构气缸动作异常
OUT TR1
AND 10.10  ; 前腔体出料夹爪气缸
ANDNOT T0232  ; 前腔体出料机械手夹爪张开位
SET W407.00  ; (I:5.06) 前腔体出料机械手夹爪张开位感应异常
LD TR1
ANDNOT 10.10  ; 前腔体出料夹爪气缸
ANDNOT T0233  ; 前腔体出料机械手夹爪夹紧位
SET W407.01  ; (I:5.07) 前腔体出料机械手夹爪夹紧位感应异常
LD TR1
ANDNOT 10.11  ; 前腔体出料升降气缸
ANDNOT T0234  ; 前腔体出料机械手升降气缸缩回位
SET W407.02  ; (I:5.08) 前腔体出料机械手升降气缸缩回位感应异常
LD TR1
AND 10.11  ; 前腔体出料升降气缸
ANDNOT T0235  ; 前腔体出料机械手升降气缸伸出位
SET W407.03  ; (I:5.09) 前腔体出料机械手升降气缸伸出位感应异常
LD TR0
!@AND T0138  ; 前下料机械手柔性报警
LD 100.02  ; 自动启动
AND 10.11  ; 前腔体出料升降气缸
OR P_On
ANDLD
SET W407.13  ; (W407.13) 前下料机械手柔性报警

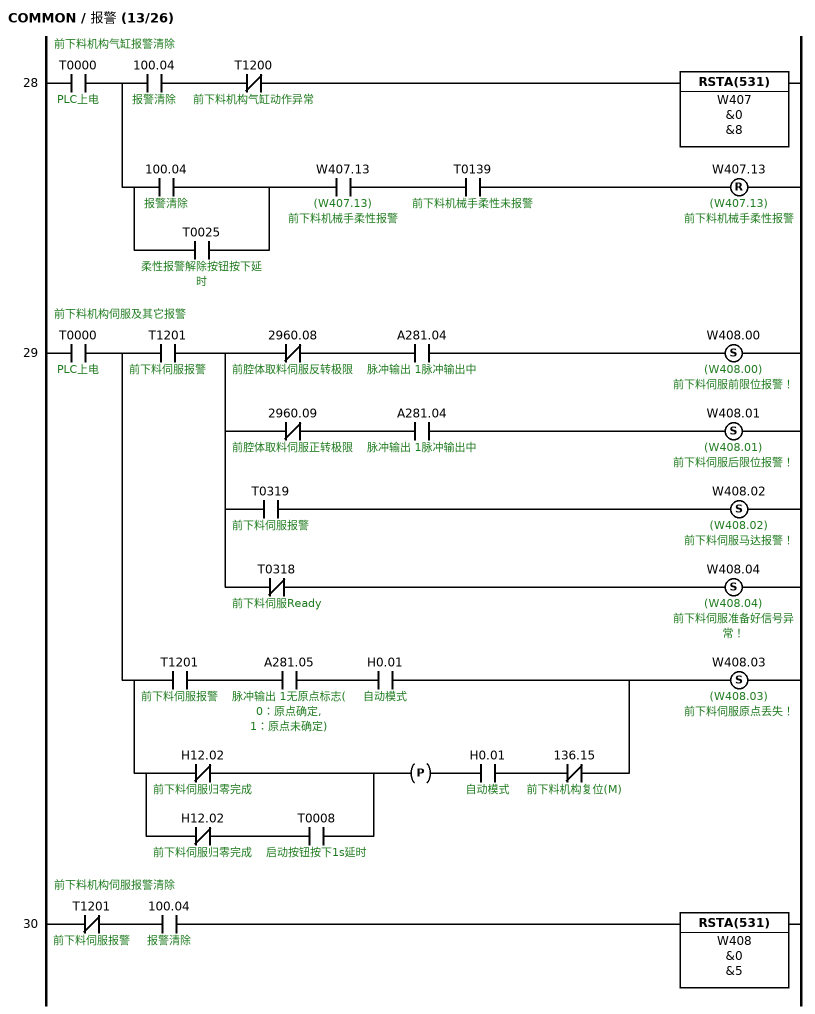
; rung 28: 前下料机构气缸报警清除
LD T0000  ; PLC上电
OUT TR0
AND 100.04  ; 报警清除
ANDNOT T1200  ; 前下料机构气缸动作异常
RSTA(531) W407 &0 &8
LD TR0
LD 100.04  ; 报警清除
OR T0025  ; 柔性报警解除按钮按下延时
ANDLD
AND W407.13  ; (W407.13) 前下料机械手柔性报警
AND T0139  ; 前下料机械手柔性未报警
RSET W407.13  ; (W407.13) 前下料机械手柔性报警
; rung 29: 前下料机构伺服及其它报警
LD T0000  ; PLC上电
OUT TR0
AND T1201  ; 前下料伺服报警
OUT TR1
ANDNOT 2960.08  ; 前腔体取料伺服反转极限
AND A281.04  ; 脉冲输出 1脉冲输出中
SET W408.00  ; (W408.00) 前下料伺服前限位报警！
LD TR1
ANDNOT 2960.09  ; 前腔体取料伺服正转极限
AND A281.04  ; 脉冲输出 1脉冲输出中
SET W408.01  ; (W408.01) 前下料伺服后限位报警！
LD TR1
AND T0319  ; 前下料伺服报警
SET W408.02  ; (W408.02) 前下料伺服马达报警！
LD TR1
ANDNOT T0318  ; 前下料伺服Ready
SET W408.04  ; (W408.04) 前下料伺服准备好信号异常！
LD TR0
LD T1201  ; 前下料伺服报警
AND A281.05  ; 脉冲输出 1无原点标志(0：原点确定,1：原点未确定)
AND H0.01  ; 自动模式
LDNOT H12.02  ; 前下料伺服归零完成
LDNOT H12.02  ; 前下料伺服归零完成
AND T0008  ; 启动按钮按下1s延时
ORLD
UP(521)
AND H0.01  ; 自动模式
ANDNOT 136.15  ; 前下料机构复位(M)
ORLD
ANDLD
SET W408.03  ; (W408.03) 前下料伺服原点丢失！
; rung 30: 前下料机构伺服报警清除
LDNOT T1201  ; 前下料伺服报警
AND 100.04  ; 报警清除
RSTA(531) W408 &0 &5

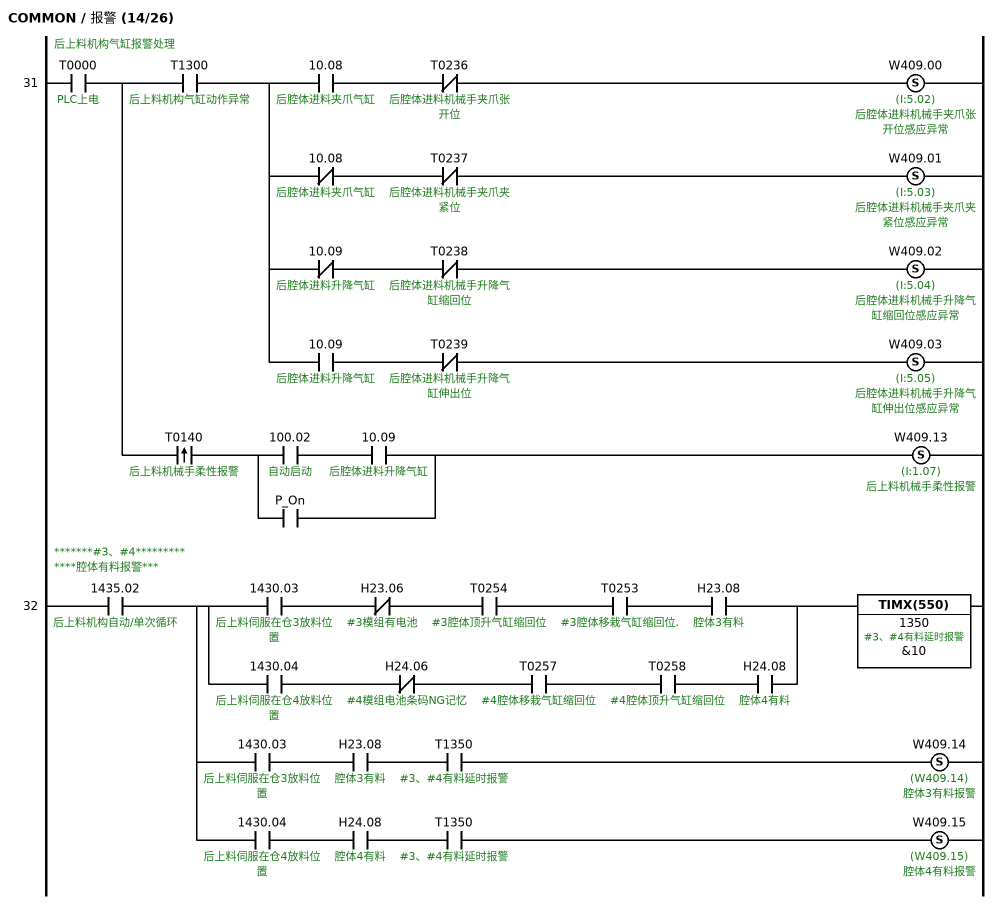
; rung 31: 后上料机构气缸报警处理
LD T0000  ; PLC上电
OUT TR0
AND T1300  ; 后上料机构气缸动作异常
OUT TR1
AND 10.08  ; 后腔体进料夹爪气缸
ANDNOT T0236  ; 后腔体进料机械手夹爪张开位
SET W409.00  ; (I:5.02) 后腔体进料机械手夹爪张开位感应异常
LD TR1
ANDNOT 10.08  ; 后腔体进料夹爪气缸
ANDNOT T0237  ; 后腔体进料机械手夹爪夹紧位
SET W409.01  ; (I:5.03) 后腔体进料机械手夹爪夹紧位感应异常
LD TR1
ANDNOT 10.09  ; 后腔体进料升降气缸
ANDNOT T0238  ; 后腔体进料机械手升降气缸缩回位
SET W409.02  ; (I:5.04) 后腔体进料机械手升降气缸缩回位感应异常
LD TR1
AND 10.09  ; 后腔体进料升降气缸
ANDNOT T0239  ; 后腔体进料机械手升降气缸伸出位
SET W409.03  ; (I:5.05) 后腔体进料机械手升降气缸伸出位感应异常
LD TR0
!@AND T0140  ; 后上料机械手柔性报警
LD 100.02  ; 自动启动
AND 10.09  ; 后腔体进料升降气缸
OR P_On
ANDLD
SET W409.13  ; (I:1.07) 后上料机械手柔性报警
; rung 32: *******#3、#4********* / ****腔体有料报警***
LD 1435.02  ; 后上料机构自动/单次循环
OUT TR0
LD 1430.03  ; 后上料伺服在仓3放料位置
ANDNOT H23.06  ; #3模组有电池
AND T0254  ; #3腔体顶升气缸缩回位
AND T0253  ; #3腔体移栽气缸缩回位.
AND H23.08  ; 腔体3有料
LD 1430.04  ; 后上料伺服在仓4放料位置
ANDNOT H24.06  ; #4模组电池条码NG记忆
AND T0257  ; #4腔体移栽气缸缩回位
AND T0258  ; #4腔体顶升气缸缩回位
AND H24.08  ; 腔体4有料
ORLD
ANDLD
TIMX(550) 1350 &10  ; #3、#4有料延时报警
LD TR0
AND 1430.03  ; 后上料伺服在仓3放料位置
AND H23.08  ; 腔体3有料
AND T1350  ; #3、#4有料延时报警
SET W409.14  ; (W409.14) 腔体3有料报警
LD TR0
AND 1430.04  ; 后上料伺服在仓4放料位置
AND H24.08  ; 腔体4有料
AND T1350  ; #3、#4有料延时报警
SET W409.15  ; (W409.15) 腔体4有料报警

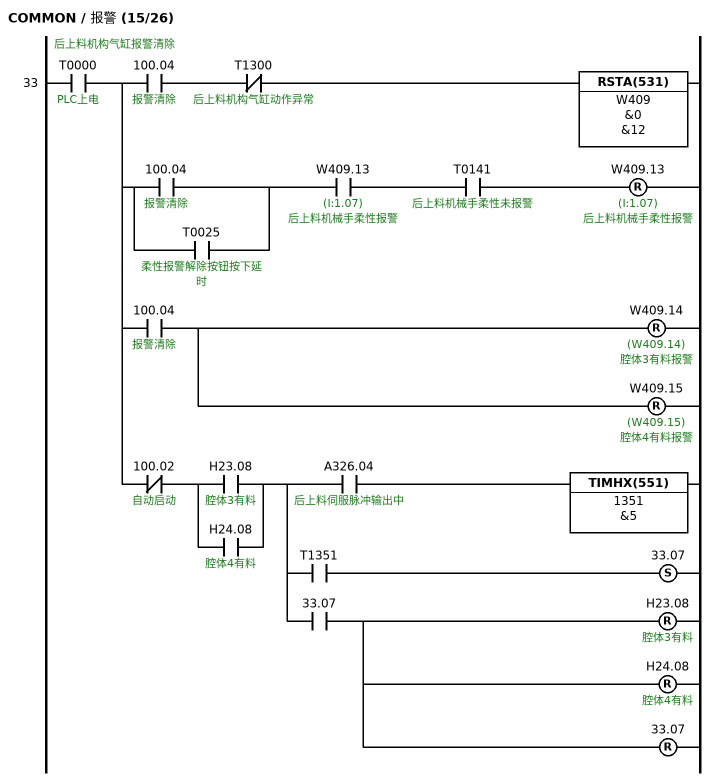
; rung 33: 后上料机构气缸报警清除
LD T0000  ; PLC上电
OUT TR0
AND 100.04  ; 报警清除
ANDNOT T1300  ; 后上料机构气缸动作异常
RSTA(531) W409 &0 &12
LD TR0
LD 100.04  ; 报警清除
OR T0025  ; 柔性报警解除按钮按下延时
ANDLD
AND W409.13  ; (I:1.07) 后上料机械手柔性报警
AND T0141  ; 后上料机械手柔性未报警
RSET W409.13  ; (I:1.07) 后上料机械手柔性报警
LD TR0
AND 100.04  ; 报警清除
RSET W409.14  ; (W409.14) 腔体3有料报警
RSET W409.15  ; (W409.15) 腔体4有料报警
LD TR0
ANDNOT 100.02  ; 自动启动
LD H23.08  ; 腔体3有料
OR H24.08  ; 腔体4有料
ANDLD
OUT TR0
AND A326.04  ; 后上料伺服脉冲输出中
TIMHX(551) 1351 &5
LD TR0
AND T1351
SET 33.07
LD TR0
AND 33.07
RSET H23.08  ; 腔体3有料
RSET H24.08  ; 腔体4有料
RSET 33.07

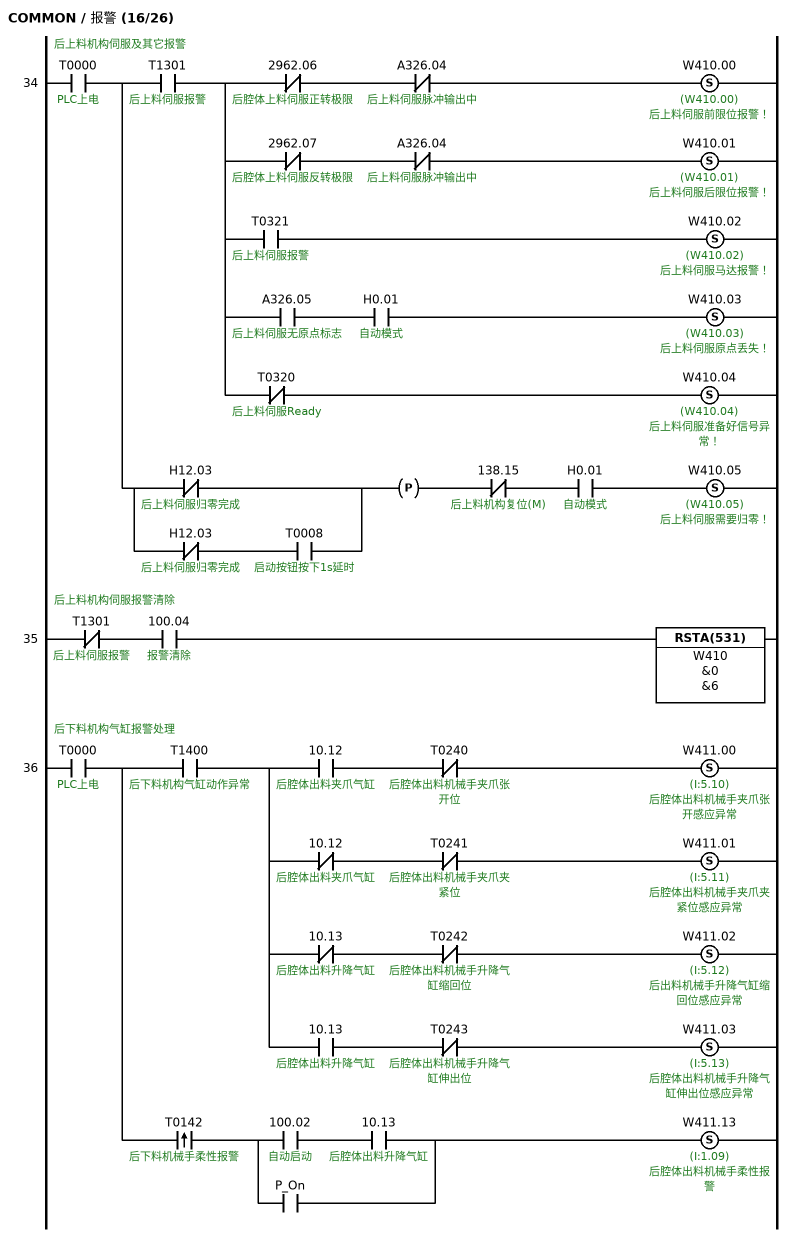
; rung 34: 后上料机构伺服及其它报警
LD T0000  ; PLC上电
OUT TR0
AND T1301  ; 后上料伺服报警
OUT TR1
ANDNOT 2962.06  ; 后腔体上料伺服正转极限
ANDNOT A326.04  ; 后上料伺服脉冲输出中
SET W410.00  ; (W410.00) 后上料伺服前限位报警！
LD TR1
ANDNOT 2962.07  ; 后腔体上料伺服反转极限
ANDNOT A326.04  ; 后上料伺服脉冲输出中
SET W410.01  ; (W410.01) 后上料伺服后限位报警！
LD TR1
AND T0321  ; 后上料伺服报警
SET W410.02  ; (W410.02) 后上料伺服马达报警！
LD TR1
AND A326.05  ; 后上料伺服无原点标志
AND H0.01  ; 自动模式
SET W410.03  ; (W410.03) 后上料伺服原点丢失！
LD TR1
ANDNOT T0320  ; 后上料伺服Ready
SET W410.04  ; (W410.04) 后上料伺服准备好信号异常！
LD TR0
LDNOT H12.03  ; 后上料伺服归零完成
LDNOT H12.03  ; 后上料伺服归零完成
AND T0008  ; 启动按钮按下1s延时
ORLD
ANDLD
UP(521)
ANDNOT 138.15  ; 后上料机构复位(M)
AND H0.01  ; 自动模式
SET W410.05  ; (W410.05) 后上料伺服需要归零！
; rung 35: 后上料机构伺服报警清除
LDNOT T1301  ; 后上料伺服报警
AND 100.04  ; 报警清除
RSTA(531) W410 &0 &6
; rung 36: 后下料机构气缸报警处理
LD T0000  ; PLC上电
OUT TR0
AND T1400  ; 后下料机构气缸动作异常
OUT TR1
AND 10.12  ; 后腔体出料夹爪气缸
ANDNOT T0240  ; 后腔体出料机械手夹爪张开位
SET W411.00  ; (I:5.10) 后腔体出料机械手夹爪张开感应异常
LD TR1
ANDNOT 10.12  ; 后腔体出料夹爪气缸
ANDNOT T0241  ; 后腔体出料机械手夹爪夹紧位
SET W411.01  ; (I:5.11) 后腔体出料机械手夹爪夹紧位感应异常
LD TR1
ANDNOT 10.13  ; 后腔体出料升降气缸
ANDNOT T0242  ; 后腔体出料机械手升降气缸缩回位
SET W411.02  ; (I:5.12) 后出料机械手升降气缸缩回位感应异常
LD TR1
AND 10.13  ; 后腔体出料升降气缸
ANDNOT T0243  ; 后腔体出料机械手升降气缸伸出位
SET W411.03  ; (I:5.13) 后腔体出料机械手升降气缸伸出位感应异常
LD TR0
!@AND T0142  ; 后下料机械手柔性报警
LD 100.02  ; 自动启动
AND 10.13  ; 后腔体出料升降气缸
OR P_On
ANDLD
SET W411.13  ; (I:1.09) 后腔体出料机械手柔性报警

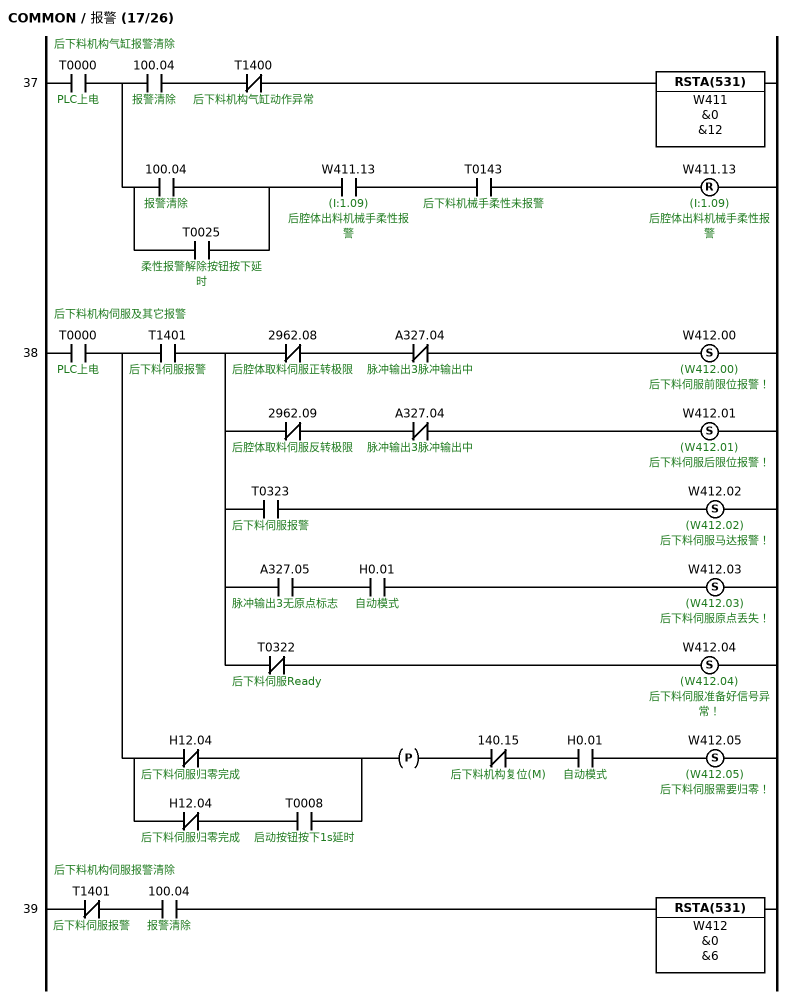
; rung 37: 后下料机构气缸报警清除
LD T0000  ; PLC上电
OUT TR0
AND 100.04  ; 报警清除
ANDNOT T1400  ; 后下料机构气缸动作异常
RSTA(531) W411 &0 &12
LD TR0
LD 100.04  ; 报警清除
OR T0025  ; 柔性报警解除按钮按下延时
ANDLD
AND W411.13  ; (I:1.09) 后腔体出料机械手柔性报警
AND T0143  ; 后下料机械手柔性未报警
RSET W411.13  ; (I:1.09) 后腔体出料机械手柔性报警
; rung 38: 后下料机构伺服及其它报警
LD T0000  ; PLC上电
OUT TR0
AND T1401  ; 后下料伺服报警
OUT TR1
ANDNOT 2962.08  ; 后腔体取料伺服正转极限
ANDNOT A327.04  ; 脉冲输出3脉冲输出中
SET W412.00  ; (W412.00) 后下料伺服前限位报警！
LD TR1
ANDNOT 2962.09  ; 后腔体取料伺服反转极限
ANDNOT A327.04  ; 脉冲输出3脉冲输出中
SET W412.01  ; (W412.01) 后下料伺服后限位报警！
LD TR1
AND T0323  ; 后下料伺服报警
SET W412.02  ; (W412.02) 后下料伺服马达报警！
LD TR1
AND A327.05  ; 脉冲输出3无原点标志
AND H0.01  ; 自动模式
SET W412.03  ; (W412.03) 后下料伺服原点丢失！
LD TR1
ANDNOT T0322  ; 后下料伺服Ready
SET W412.04  ; (W412.04) 后下料伺服准备好信号异常！
LD TR0
LDNOT H12.04  ; 后下料伺服归零完成
LDNOT H12.04  ; 后下料伺服归零完成
AND T0008  ; 启动按钮按下1s延时
ORLD
ANDLD
UP(521)
ANDNOT 140.15  ; 后下料机构复位(M)
AND H0.01  ; 自动模式
SET W412.05  ; (W412.05) 后下料伺服需要归零！
; rung 39: 后下料机构伺服报警清除
LDNOT T1401  ; 后下料伺服报警
AND 100.04  ; 报警清除
RSTA(531) W412 &0 &6

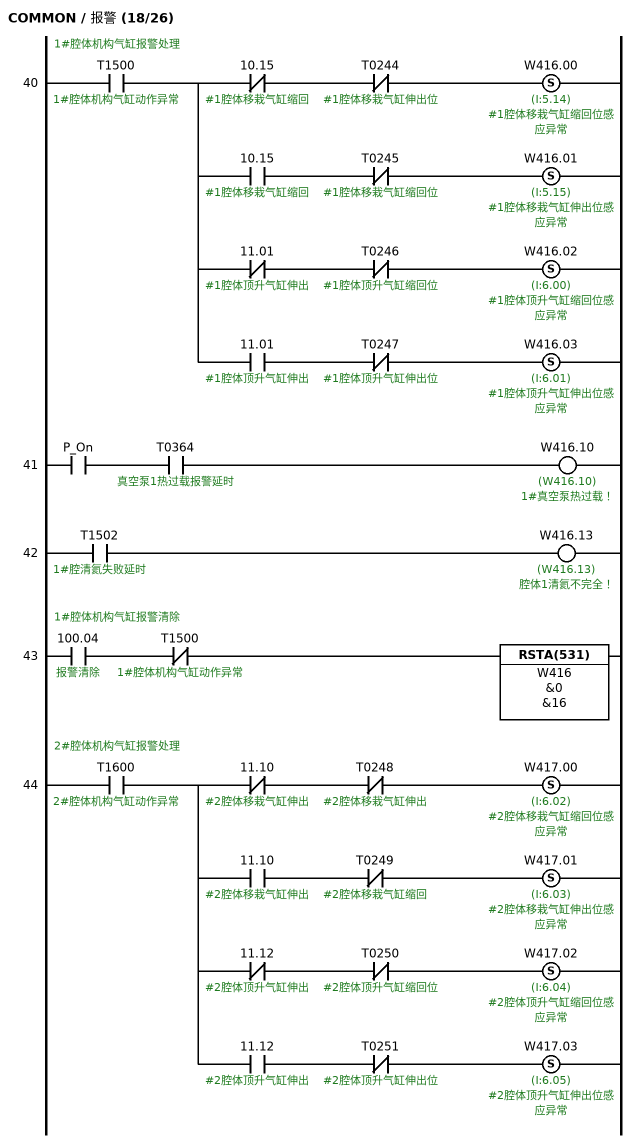
; rung 40: 1#腔体机构气缸报警处理
LD T1500  ; 1#腔体机构气缸动作异常
OUT TR0
ANDNOT 10.15  ; #1腔体移栽气缸缩回
ANDNOT T0244  ; #1腔体移栽气缸伸出位
SET W416.00  ; (I:5.14) #1腔体移栽气缸缩回位感应异常
LD TR0
AND 10.15  ; #1腔体移栽气缸缩回
ANDNOT T0245  ; #1腔体移栽气缸缩回位
SET W416.01  ; (I:5.15) #1腔体移栽气缸伸出位感应异常
LD TR0
ANDNOT 11.01  ; #1腔体顶升气缸伸出
ANDNOT T0246  ; #1腔体顶升气缸缩回位
SET W416.02  ; (I:6.00) #1腔体顶升气缸缩回位感应异常
LD TR0
AND 11.01  ; #1腔体顶升气缸伸出
ANDNOT T0247  ; #1腔体顶升气缸伸出位
SET W416.03  ; (I:6.01) #1腔体顶升气缸伸出位感应异常
; rung 41
LD P_On
AND T0364  ; 真空泵1热过载报警延时
OUT W416.10  ; (W416.10) 1#真空泵热过载！
; rung 42
LD T1502  ; 1#腔清氦失败延时
OUT W416.13  ; (W416.13) 腔体1清氦不完全！
; rung 43: 1#腔体机构气缸报警清除
LD 100.04  ; 报警清除
ANDNOT T1500  ; 1#腔体机构气缸动作异常
RSTA(531) W416 &0 &16
; rung 44: 2#腔体机构气缸报警处理
LD T1600  ; 2#腔体机构气缸动作异常
OUT TR0
ANDNOT 11.10  ; #2腔体移栽气缸伸出
ANDNOT T0248  ; #2腔体移栽气缸伸出
SET W417.00  ; (I:6.02) #2腔体移栽气缸缩回位感应异常
LD TR0
AND 11.10  ; #2腔体移栽气缸伸出
ANDNOT T0249  ; #2腔体移栽气缸缩回
SET W417.01  ; (I:6.03) #2腔体移栽气缸伸出位感应异常
LD TR0
ANDNOT 11.12  ; #2腔体顶升气缸伸出
ANDNOT T0250  ; #2腔体顶升气缸缩回位
SET W417.02  ; (I:6.04) #2腔体顶升气缸缩回位感应异常
LD TR0
AND 11.12  ; #2腔体顶升气缸伸出
ANDNOT T0251  ; #2腔体顶升气缸伸出位
SET W417.03  ; (I:6.05) #2腔体顶升气缸伸出位感应异常

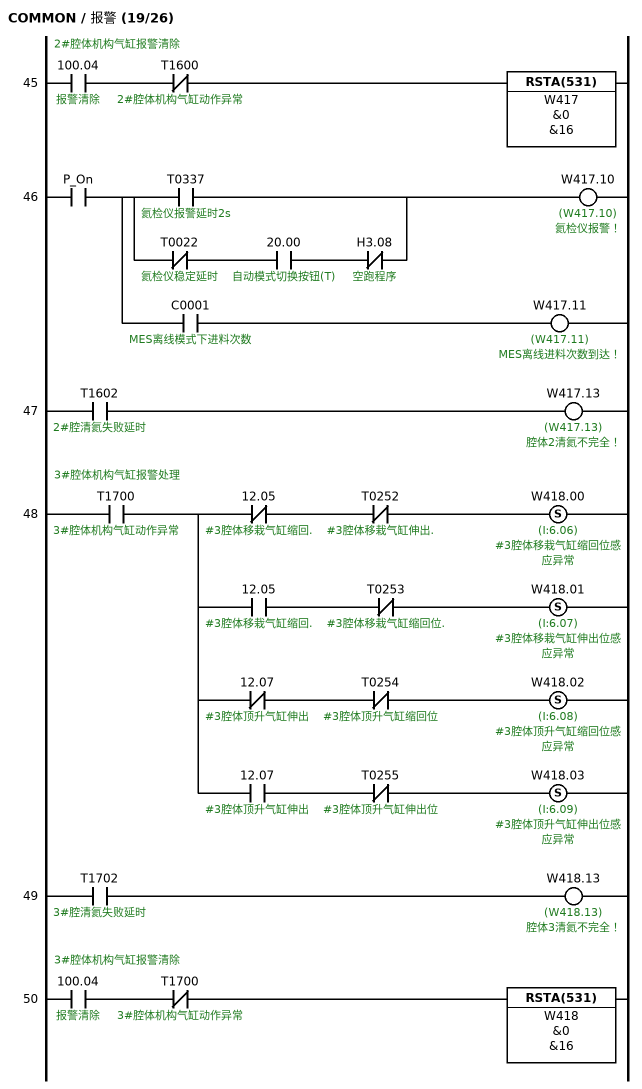
; rung 45: 2#腔体机构气缸报警清除
LD 100.04  ; 报警清除
ANDNOT T1600  ; 2#腔体机构气缸动作异常
RSTA(531) W417 &0 &16
; rung 46
LD P_On
OUT TR0
LD T0337  ; 氦检仪报警延时2s
LDNOT T0022  ; 氦检仪稳定延时
AND 20.00  ; 自动模式切换按钮(T)
ANDNOT H3.08  ; 空跑程序
ORLD
ANDLD
OUT W417.10  ; (W417.10) 氦检仪报警！
LD TR0
AND C0001  ; MES离线模式下进料次数
OUT W417.11  ; (W417.11) MES离线进料次数到达！
; rung 47
LD T1602  ; 2#腔清氦失败延时
OUT W417.13  ; (W417.13) 腔体2清氦不完全！
; rung 48: 3#腔体机构气缸报警处理
LD T1700  ; 3#腔体机构气缸动作异常
OUT TR0
ANDNOT 12.05  ; #3腔体移栽气缸缩回.
ANDNOT T0252  ; #3腔体移栽气缸伸出.
SET W418.00  ; (I:6.06) #3腔体移栽气缸缩回位感应异常
LD TR0
AND 12.05  ; #3腔体移栽气缸缩回.
ANDNOT T0253  ; #3腔体移栽气缸缩回位.
SET W418.01  ; (I:6.07) #3腔体移栽气缸伸出位感应异常
LD TR0
ANDNOT 12.07  ; #3腔体顶升气缸伸出
ANDNOT T0254  ; #3腔体顶升气缸缩回位
SET W418.02  ; (I:6.08) #3腔体顶升气缸缩回位感应异常
LD TR0
AND 12.07  ; #3腔体顶升气缸伸出
ANDNOT T0255  ; #3腔体顶升气缸伸出位
SET W418.03  ; (I:6.09) #3腔体顶升气缸伸出位感应异常
; rung 49
LD T1702  ; 3#腔清氦失败延时
OUT W418.13  ; (W418.13) 腔体3清氦不完全！
; rung 50: 3#腔体机构气缸报警清除
LD 100.04  ; 报警清除
ANDNOT T1700  ; 3#腔体机构气缸动作异常
RSTA(531) W418 &0 &16

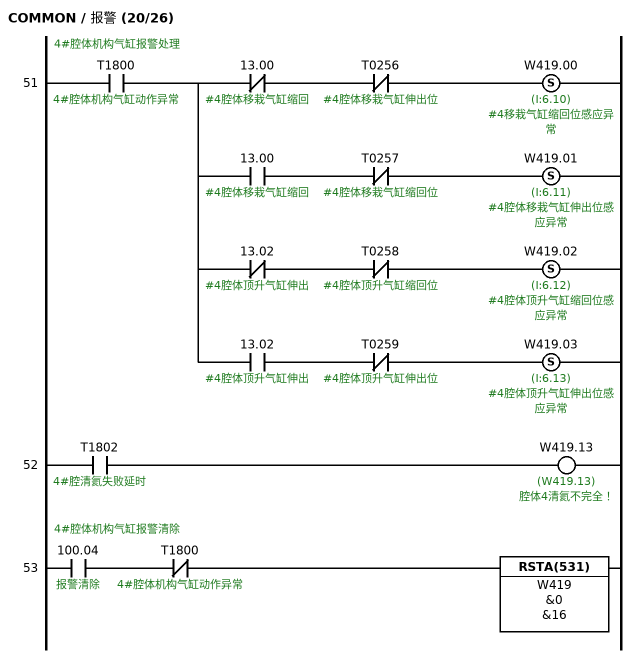
; rung 51: 4#腔体机构气缸报警处理
LD T1800  ; 4#腔体机构气缸动作异常
OUT TR0
ANDNOT 13.00  ; #4腔体移栽气缸缩回
ANDNOT T0256  ; #4腔体移栽气缸伸出位
SET W419.00  ; (I:6.10) #4移栽气缸缩回位感应异常
LD TR0
AND 13.00  ; #4腔体移栽气缸缩回
ANDNOT T0257  ; #4腔体移栽气缸缩回位
SET W419.01  ; (I:6.11) #4腔体移栽气缸伸出位感应异常
LD TR0
ANDNOT 13.02  ; #4腔体顶升气缸伸出
ANDNOT T0258  ; #4腔体顶升气缸缩回位
SET W419.02  ; (I:6.12) #4腔体顶升气缸缩回位感应异常
LD TR0
AND 13.02  ; #4腔体顶升气缸伸出
ANDNOT T0259  ; #4腔体顶升气缸伸出位
SET W419.03  ; (I:6.13) #4腔体顶升气缸伸出位感应异常
; rung 52
LD T1802  ; 4#腔清氦失败延时
OUT W419.13  ; (W419.13) 腔体4清氦不完全！
; rung 53: 4#腔体机构气缸报警清除
LD 100.04  ; 报警清除
ANDNOT T1800  ; 4#腔体机构气缸动作异常
RSTA(531) W419 &0 &16

